(* IEC 61131-3 sources: LASAL/Class/CommandRouter, 1 file *)

(* ---- CommandRouter.st ---- *)
(*!
<Class
	Name               = "CommandRouter"
	Revision           = "0.0"
	RealtimeTask       = "false"
	CyclicTask         = "false"
	BackgroundTask     = "false"
	Sigmatek           = "false"
	OSInterface        = "false"
	HighPriority       = "false"
	Automatic          = "false"
	UpdateMode         = "Prescan"
	SharedCommandTable = "true"
	Objectsize         = "(480,120)">
	<Channels>
		<Server Name="Acc" Visualized="false" Initialize="true" WriteProtected="false" Retentive="SRam"/>
		<Server Name="CmdRouter" Visualized="false" Initialize="false" WriteProtected="true" Retentive="false"/>
		<Server Name="Debug" Visualized="false" Initialize="false" WriteProtected="true" Retentive="false"/>
		<Server Name="Speed" Visualized="false" Initialize="true" WriteProtected="false" Retentive="SRam"/>
		<Server Name="YAcc" Visualized="false" Initialize="true" WriteProtected="false" Retentive="SRam"/>
		<Server Name="YSpeed" Visualized="false" Initialize="true" WriteProtected="false" Retentive="SRam"/>
		<Client Name="clib" Required="false" Internal="false"/>
		<Client Name="Controller" Required="true" Internal="false"/>
	</Channels>
</Class>
*)
CommandRouter : CLASS
  //Servers:
	CmdRouter 	: SvrChCmd_DINT;
	Debug 	: SvrCh_DINT;
	Speed 	: SvrCh_DINT;
	Acc 	: SvrCh_DINT;
	YSpeed 	: SvrCh_DINT;
	YAcc 	: SvrCh_DINT;
  //Clients:
	Controller 	: CltChCmd_MoveController;
	clib 	: CltChCmd_SigCLib;
  //Variables:
		DataBuffer : ARRAY [0..1024] OF CHAR;

		Command : ARRAY [0..8] OF CHAR;

		X : ARRAY [0..8] OF CHAR;

		Y : ARRAY [0..8] OF CHAR;

		Phi : ARRAY [0..8] OF CHAR;

  //Functions:

	FUNCTION GLOBAL SetData
		VAR_INPUT
			pData 	: ^void;
			size 	: UDINT;
		END_VAR;
  //Tables:
	FUNCTION @STD
		VAR_OUTPUT
			ret_code	: CONFSTATES;
		END_VAR;
	FUNCTION GLOBAL TAB @CT_;
END_CLASS;

#pragma usingLtd MoveController
#pragma usingLtd SigCLib

(* CommandRouter::SetData
Allows the tcp server to write the received data into the commandRouter instances
data buffer.
Appends a 0 at the end of the received string as string termination.
*)
FUNCTION GLOBAL CommandRouter::SetData
	VAR_INPUT
    // pointer to the data
		pData 	: ^void;
    // size of the received data
		size 	: UDINT;
	END_VAR

  VAR
    pString : ^CHAR;
  	counter : DINT;
    commandSize : DINT;
    parameterSize : DINT;
    XVal : DINT;
    YVal : DINT;
    ZVal : DINT;
    PhiVal : DINT;
  END_VAR

  // size of the parameter plus one semicolon
  parameterSize := 8 + 1;

  Debug += 1;

  _memcpy(ptr1:=#DataBuffer[0], ptr2:=pData, cntr:=size);
  DataBuffer[size] := 0;
  pString := #DataBuffer[0];

  // get first 5 values (this represents the command)
  _memcpy(ptr1:=#Command, ptr2:=pString, cntr:=8);

  // get the other values depending
  // on the command (these represent the command parameters)
  if clib.StrCmp(ps1:=#Command[0], ps2:="CMOVEABS") = 0 then
    _memcpy(ptr1:=#X, ptr2:=pString+parameterSize, cntr:=8);
    _memcpy(ptr1:=#Y, ptr2:=pString+parameterSize*2, cntr:=8);
    _memcpy(ptr1:=#Phi, ptr2:=pString+parameterSize*3, cntr:=8);

    XVal := clib.AToI(ps1:=#X[0]);
    YVal := clib.AToI(ps1:=#Y[0]);
    PhiVal := cLib.AToI(ps1:=#Phi[0]);

    Controller.MoveAxis(XPos:=XVal, YPos:=YVal, Speed:=Speed, Accel:=Acc, YSpeed:=YSpeed, YAcc:=YAcc);

  ELSIF clib.StrCmp(ps1:=#Command[0], ps2:="CPOWERON") = 0 then
    Controller.TogglePower(Power:=1);
    ELSIF clib.StrCmp(ps1:=#Command[0], ps2:="CPOWEROF") = 0 then
    Controller.TogglePower(Power:=0);
  end_if;

END_FUNCTION
